FUNCTION_BLOCK PressureGradient
VAR_INPUT
	TotalVolume: LREAL;
	BulkModulus: LREAL;
	FlowrateIn: LREAL;
	FlowrateOut: LREAL;
	pMax : LREAL;
	p0 : LREAL;
	param : ST_pValveControlledCylinder;
END_VAR
VAR_OUTPUT
	PressureGradient : LREAL;
	Pressure : LREAL;
END_VAR
VAR
	ssMethodType : SINT := 1; 
	fbPressurePascal : DiscreteTimeIntegrator_Init;
END_VAR

 
//PressureGradient in [Pascal/s]
PressureGradient := (FlowrateIn - FlowrateOut) * (BulkModulus / TotalVolume);


//Pressure in [Pascal]
fbPressurePascal(
	ssMethodType := ssMethodType,
	tCycle := param.tCycle,
	In := PressureGradient,
	Init := p0,
	minOut := G_ActuationSystems.ReturnPressure,
	maxOut := param.pAmax,
	Out => Pressure
	);

END_FUNCTION_BLOCK

(* stored: Version 1.1.0.1, ProductVersion 3.1.4024.9
   POU PressureGradient: Id {0ae25e94-6017-429e-9462-38875999b492}, SpecialFunc None *)
